// TwinCAT 3 PLC project struckig_unittest
// ProgramVersion: 3.1.4024.12
// libraries:
//   Struckig, * (Struckig)
//   Tc2_Standard, * (Beckhoff Automation GmbH)
//   Tc2_System, * (Beckhoff Automation GmbH)
//   Tc3_Module, * (Beckhoff Automation GmbH)
//   TcUnit, * (www.tcunit.org)
// project tree:
//   / PlcTask.TcTTO (not stored)
//   POUs/ run_and_return_duration.TcPOU, KnownExamplesTest.TcPOU, MAIN.TcPOU
// real-time tasks:
//   TASK PlcTask: cycle T#10ms, priority 20, ADS port 350

// ---- POUs/run_and_return_duration.TcPOU
FUNCTION run_and_return_duration : LREAL
VAR_INPUT
  ruckig : REFERENCE TO Struckig.Ruckig;
  input : REFERENCE TO Struckig.InputParameter;
  output : REFERENCE TO Struckig.OutputParameter;  
END_VAR

WHILE(ruckig.update(input, output) = Struckig.StateEnum.busy)
DO
  input.current_position := output.new_position;
  input.current_velocity := output.new_velocity;
  input.current_acceleration := output.new_acceleration;
END_WHILE

run_and_return_duration := output.trajectory.duration;

END_FUNCTION

// ---- POUs/KnownExamplesTest.TcPOU
FUNCTION_BLOCK KnownExamplesTest EXTENDS TcUnit.FB_TestSuite

example01();
example02();
example03();
example05();
example06();
example07();
example08();
example09();
example10();
example11();
example12();
example13();
example14();
example15();
example16();
example17();
example18();

METHOD example01
VAR_INST
  ruckig : Struckig.Ruckig(0.005);
  input : Struckig.InputParameter(3) := (
    synchronizationType := SynchronizationTypeEnum.none,        
    max_velocity :=         [ 1.0, 1.0, 1.0 ],
    max_acceleration :=     [ 1.0, 1.0, 1.0 ],
    max_jerk :=             [ 1.0, 1.0, 1.0 ],
    current_position :=     [ 0.0, 0.0, 0.0 ],
    current_velocity :=     [ 0.0, 0.0, 0.0 ],
    current_acceleration := [ 0.0, 0.0, 0.0 ],
    target_position :=      [ 0.0, 0.0, 0.0 ],
    target_velocity :=      [ 0.0, 0.0, 0.0 ],
    target_acceleration :=  [ 0.0, 0.0, 0.0 ]
  );
  output : Struckig.OutputParameter;
END_VAR
TEST('Example-01');

AssertEquals_LREAL(Expected := 0.0,
             Actual := run_and_return_duration(ruckig, input, output),
             DELTA := 1E-8,
             Message := '');
 
TEST_FINISHED();
END_METHOD

METHOD example02
VAR_INST
  ruckig : Struckig.Ruckig(0.005);
  input : Struckig.InputParameter(3) := (
    synchronizationType := SynchronizationTypeEnum.none,        
    max_velocity :=         [ 1.0, 1.0, 1.0 ],
    max_acceleration :=     [ 1.0, 1.0, 1.0 ],
    max_jerk :=             [ 1.0, 1.0, 1.0 ],
    current_position :=     [ 0.0, 0.0, 0.0 ],
    current_velocity :=     [ 0.0, 0.0, 0.0 ],
    current_acceleration := [ 0.0, 0.0, 0.0 ],
    target_position :=      [ 0.0, 1E-17, -1E-17 ],
    target_velocity :=      [ 0.0, 0.0, 0.0 ],
    target_acceleration :=  [ 0.0, 0.0, 0.0 ]
  );
  output : Struckig.OutputParameter;  
END_VAR
TEST('Example-02');

AssertEquals_LREAL(Expected := 1E-18,
             Actual := run_and_return_duration(ruckig, input, output),
             Delta := 1E-19,
             Message := '');
 
TEST_FINISHED();
END_METHOD

METHOD example03
VAR_INST
  ruckig : Struckig.Ruckig(0.005);
  input : Struckig.InputParameter(3) := (
    synchronizationType := SynchronizationTypeEnum.none,        
    max_velocity :=         [ 1.0, 1.0, 1.0 ],
    max_acceleration :=     [ 1.0, 1.0, 1.0 ],
    max_jerk :=             [ 1.0, 1.0, 1.0 ],
    current_position :=     [ 0.0, 1E-17, -1E-17 ],
    current_velocity :=     [ 0.0, 0.0, 0.0 ],
    current_acceleration := [ 0.0, 0.0, 0.0 ],
    target_position :=      [ 1.0, 1.0, 1.0 ],
    target_velocity :=      [ 0.0, 0.0, 0.0 ],
    target_acceleration :=  [ 0.0, 0.0, 0.0 ]
  );
  output : Struckig.OutputParameter;
  
END_VAR
TEST('Example-03');

AssertEquals_LREAL(Expected := 3.1748021039,
             Actual := run_and_return_duration(ruckig, input, output),
             DELTA := 1E-8,
             Message := '');
 
TEST_FINISHED();
END_METHOD

METHOD example04
VAR_INST
  ruckig : Struckig.Ruckig(0.005);
  input : Struckig.InputParameter(3) := (
    synchronizationType := SynchronizationTypeEnum.none,        
    max_velocity :=         [ 1.0, 1.0, 1.0 ],
    max_acceleration :=     [ 1.0, 1.0, 1.0 ],
    max_jerk :=             [ 2.0, 2.0, 2.0 ],
    current_position :=     [ 0.0, 0.0, 0.0 ],
    current_velocity :=     [ 0.0, 0.0, 0.0 ],
    current_acceleration := [ 0.0, 0.0, 0.0 ],
    target_position :=      [ 1.0, 1.0, 1.0 ],
    target_velocity :=      [ 0.0, 0.0, 0.0 ],
    target_acceleration :=  [ 0.0, 0.0, 0.0 ]
  );
  output : Struckig.OutputParameter;
  
END_VAR
TEST('Example-04');

AssertEquals_LREAL(Expected := 2.5615528128,
             Actual := run_and_return_duration(ruckig, input, output),
             DELTA := 1E-8,
             Message := '');
 
TEST_FINISHED();
END_METHOD

METHOD example05
VAR_INST
  ruckig : Struckig.Ruckig(0.005);
  input : Struckig.InputParameter(3) := (
    synchronizationType := SynchronizationTypeEnum.none,        
    max_velocity :=         [ 0.6, 0.6, 0.6 ],
    max_acceleration :=     [ 1.0, 1.0, 1.0 ],
    max_jerk :=             [ 2.0, 2.0, 2.0 ],
    current_position :=     [ 0.0, 0.0, 0.0 ],
    current_velocity :=     [ 0.0, 0.0, 0.0 ],
    current_acceleration := [ 0.0, 0.0, 0.0 ],
    target_position :=      [ 1.0, 1.0, 1.0 ],
    target_velocity :=      [ 0.0, 0.0, 0.0 ],
    target_acceleration :=  [ 0.0, 0.0, 0.0 ]
  );
  output : Struckig.OutputParameter;
  
END_VAR
TEST('Example-05');

AssertEquals_LREAL(Expected := 2.7666666667,
             Actual := run_and_return_duration(ruckig, input, output),
             DELTA := 1E-8,
             Message := '');
 
TEST_FINISHED();
END_METHOD

METHOD example06
VAR_INST
  ruckig : Struckig.Ruckig(0.005);
  input : Struckig.InputParameter(3) := (
    synchronizationType := SynchronizationTypeEnum.none,        
    max_velocity :=         [ 0.4, 0.4, 0.4 ],
    max_acceleration :=     [ 1.0, 1.0, 1.0 ],
    max_jerk :=             [ 2.0, 2.0, 2.0 ],
    current_position :=     [ 0.0, 0.0, 0.0 ],
    current_velocity :=     [ 0.0, 0.0, 0.0 ],
    current_acceleration := [ 0.0, 0.0, 0.0 ],
    target_position :=      [ 1.0, 1.0, 1.0 ],
    target_velocity :=      [ 0.0, 0.0, 0.0 ],
    target_acceleration :=  [ 0.0, 0.0, 0.0 ]
  );
  output : Struckig.OutputParameter;
  
END_VAR
TEST('Example-06');

AssertEquals_LREAL(Expected := 3.394427191,
             Actual := run_and_return_duration(ruckig, input, output),
             DELTA := 1E-8,
             Message := '');
 
TEST_FINISHED();
END_METHOD

METHOD example07
VAR_INST
  ruckig : Struckig.Ruckig(0.005);
  input : Struckig.InputParameter(3) := (
    synchronizationType := SynchronizationTypeEnum.none,        
    max_velocity :=         [ 1.0, 1.0, 1.0 ],
    max_acceleration :=     [ 1.0, 1.0, 1.0 ],
    max_jerk :=             [ 2.0, 2.0, 2.0 ],
    current_position :=     [ 0.0, 0.0, 0.0 ],
    current_velocity :=     [ 0.3, 0.3, 0.3 ],
    current_acceleration := [ 0.0, 0.0, 0.0 ],
    target_position :=      [ 1.0, 1.0, 1.0 ],
    target_velocity :=      [ 0.0, 0.0, 0.0 ],
    target_acceleration :=  [ 0.0, 0.0, 0.0 ]
  );
  output : Struckig.OutputParameter;
  
END_VAR
TEST('Example-07');

AssertEquals_LREAL(Expected := 2.2319602829,
             Actual := run_and_return_duration(ruckig, input, output),
             DELTA := 1E-8,
             Message := '');
 
TEST_FINISHED();
END_METHOD

METHOD example08
VAR_INST
  ruckig : Struckig.Ruckig(0.005);
  input : Struckig.InputParameter(3) := (
    synchronizationType := SynchronizationTypeEnum.none,        
    max_velocity :=         [ 0.6, 0.6, 0.6 ],
    max_acceleration :=     [ 1.0, 1.0, 1.0 ],
    max_jerk :=             [ 2.0, 2.0, 2.0 ],
    current_position :=     [ 0.0, 0.0, 0.0 ],
    current_velocity :=     [ 0.3, 0.3, 0.3 ],
    current_acceleration := [ 0.0, 0.0, 0.0 ],
    target_position :=      [ 1.0, 1.0, 1.0 ],
    target_velocity :=      [ 0.0, 0.0, 0.0 ],
    target_acceleration :=  [ 0.0, 0.0, 0.0 ]
  );
  output : Struckig.OutputParameter;
  
END_VAR
TEST('Example-08');

AssertEquals_LREAL(Expected := 2.410315834,
             Actual := run_and_return_duration(ruckig, input, output),
             DELTA := 1E-8,
             Message := '');
 
TEST_FINISHED();
END_METHOD

METHOD example09
VAR_INST
  ruckig : Struckig.Ruckig(0.005);
  input : Struckig.InputParameter(3) := (
    synchronizationType := SynchronizationTypeEnum.none,        
    max_velocity :=         [ 0.6, 0.6, 0.6 ],
    max_acceleration :=     [ 1.0, 1.0, 1.0 ],
    max_jerk :=             [ 2.0, 2.0, 2.0 ],
    current_position :=     [ 0.0, 0.0, 0.0 ],
    current_velocity :=     [ 0.0, 0.0, 0.0 ],
    current_acceleration := [ 0.0, 0.0, 0.0 ],
    target_position :=      [ -1.0, -1.0, -1.0 ],
    target_velocity :=      [ 0.0, 0.0, 0.0 ],
    target_acceleration :=  [ 0.0, 0.0, 0.0 ]
  );
  output : Struckig.OutputParameter;
  
END_VAR
TEST('Example-09');

AssertEquals_LREAL(Expected := 2.7666666667,
             Actual := run_and_return_duration(ruckig, input, output),
             DELTA := 1E-8,
             Message := '');
 
TEST_FINISHED();
END_METHOD

METHOD example10
VAR_INST
  ruckig : Struckig.Ruckig(0.005);
  input : Struckig.InputParameter(3) := (
    synchronizationType := SynchronizationTypeEnum.none,        
    max_velocity :=         [ 10.0, 10.0, 10.0 ],
    max_acceleration :=     [ 10.0, 10.0, 10.0 ],
    max_jerk :=             [ 2.0, 2.0, 2.0 ],
    current_position :=     [ 0.0, 0.0, 0.0 ],
    current_velocity :=     [ 0.2, 0.2, 0.2 ],
    current_acceleration := [ 0.0, 0.0, 0.0 ],
    target_position :=      [ -1.0, -1.0, -1.0 ],
    target_velocity :=      [ 0.0, 0.0, 0.0 ],
    target_acceleration :=  [ 0.0, 0.0, 0.0 ]
  );
  output : Struckig.OutputParameter;
  
END_VAR
TEST('Example-10');

AssertEquals_LREAL(Expected := 2.7338531701,
             Actual := run_and_return_duration(ruckig, input, output),
             DELTA := 1E-8,
             Message := '');
 
TEST_FINISHED();
END_METHOD

METHOD example11
VAR_INST
  ruckig : Struckig.Ruckig(0.005);
  input : Struckig.InputParameter(3) := (
    synchronizationType := SynchronizationTypeEnum.none,        
    max_velocity :=         [ 0.4, 0.4, 0.4 ],
    max_acceleration :=     [ 1.0, 1.0, 1.0 ],
    max_jerk :=             [ 2.0, 2.0, 2.0 ],
    current_position :=     [ -1.0, -1.0, -1.0 ],
    current_velocity :=     [ 0.2, 0.2, 0.2 ],
    current_acceleration := [ 0.0, 0.0, 0.0 ],
    target_position :=      [ 1.0, 1.0, 1.0 ],
    target_velocity :=      [ 0.0, 0.0, 0.0 ],
    target_acceleration :=  [ 0.0, 0.0, 0.0 ]
  );
  output : Struckig.OutputParameter;
  
END_VAR
TEST('Example-11');

AssertEquals_LREAL(Expected := 5.6053274785,
             Actual := run_and_return_duration(ruckig, input, output),
             DELTA := 1E-8,
             Message := '');
 
TEST_FINISHED();
END_METHOD

METHOD example12
VAR_INST
  ruckig : Struckig.Ruckig(0.005);
  input : Struckig.InputParameter(3) := (
    synchronizationType := SynchronizationTypeEnum.none,        
    max_velocity :=         [ 3.0, 3.0, 3.0 ],
    max_acceleration :=     [ 0.5, 0.5, 0.5 ],
    max_jerk :=             [ 0.2, 0.2, 0.2 ],
    current_position :=     [ 0.3888899206957 - 10E-14, 0.0, 0.0 ],
    current_velocity :=     [ 0.2231429352410215, 0.0, 0.0 ],
    current_acceleration := [ -0.2987593916455, 0.0, 0.0 ],
    target_position :=      [ 0.5, 0.0, 0.0 ],
    target_velocity :=      [ 0.0, 0.0, 0.0 ],
    target_acceleration :=  [ 0.0, 0.0, 0.0 ]
  );
  output : Struckig.OutputParameter;
  
END_VAR
TEST('Example-12');

AssertEquals_LREAL(Expected := 1.4939456041,
             Actual := run_and_return_duration(ruckig, input, output),
             DELTA := 1E-8,
             Message := '');
 
TEST_FINISHED();
END_METHOD

METHOD example13
VAR_INST
  ruckig : Struckig.Ruckig(0.005);
  input : Struckig.InputParameter(3) := (
    synchronizationType := SynchronizationTypeEnum.none,        
    max_velocity :=         [ 12.9892953062198, 3.74169932927481, 1.42398447457303 ],
    max_acceleration :=     [ 4.2162106624246, 10.2906731766853, 2.1869079548297 ],
    max_jerk :=             [ 8.03496976453435, 0.200684346397485 - 1.0E-14, 0.0848503482861296 ],
    current_position :=     [ -5.54640573838539, -2.34195463203842, 5.10070661762967 ],
    current_velocity :=     [ 0.824843228617216, -1.03863337183304, -0.749451523227729 ],
    current_acceleration := [ -0.119403564898501, 0.923861820607788, 3.04022341347259 ],
    target_position :=      [ -1.58293112753888, 0.383405919465141, 5.79349604610299 ],
    target_velocity :=      [ -1.59453676324393, 0.0, -0.0693173526513803 ],
    target_acceleration :=  [ -0.664429703711622, 0.0, 0.0 ]
  );
  output : Struckig.OutputParameter;
  
END_VAR
TEST('Example-13');

AssertEquals_LREAL(Expected := 1921.0797627836,
             Actual := run_and_return_duration(ruckig, input, output),
             DELTA := 1E-8,
             Message := '');
 
TEST_FINISHED();
END_METHOD

METHOD example14
VAR_INST
  ruckig : Struckig.Ruckig(0.005);
  input : Struckig.InputParameter(3) := (
    synchronizationType := SynchronizationTypeEnum.none,        
    max_velocity :=         [ 8.65978706670502, 5.94921088330542, 10.7652253566829 ],
    max_acceleration :=     [ 3.40137210377608, 4.04166318018487, 10.8617860610581 ],
    max_jerk :=             [ 10.9542353113865, 3.11056302676629, 0.798055744482636 + 9e-12 ],
    current_position :=     [ -6.49539540831446, 6.14883133273172, -2.02636240900911 ],
    current_velocity :=     [ -1.14327601654428, 0.00991019970085593, -1.00932863927626 ],
    current_acceleration := [ -1.73501068960131, -0.584885092422228, 0 ],
    target_position :=      [ 4.4676187540058, 2.93367894961155, -0.646008452514058 ],
    target_velocity :=      [ -0.544559915133859, 0.298517792372943, 1.6058847848484 ],
    target_acceleration :=  [ -1.31832055647831, 0, 0 ]
  );
  output : Struckig.OutputParameter;
  
END_VAR
TEST('Example-14');

AssertEquals_LREAL(Expected := 4.6277455678,
             Actual := run_and_return_duration(ruckig, input, output),
             DELTA := 1E-8,
             Message := '');
 
TEST_FINISHED();
END_METHOD

METHOD example15
VAR_INST
  ruckig : Struckig.Ruckig(0.005);
  input : Struckig.InputParameter(3) := (
    synchronizationType := SynchronizationTypeEnum.none,        
    max_velocity :=         [ 7.97399137456765, 2.68591430972239, 9.54987666746364 ],
    max_acceleration :=     [ 5.44679859206862, 7.61752909348119, 0.473482772614085 ],
    max_jerk :=             [ 7.88958080921515, 5.26855927512131, 0.764061581326592 - 1e-14 ],
    current_position :=     [ 7.06378251402596, -2.4834697862831, -0.843847405371359 ],
    current_velocity :=     [ 0.436985859305842, 0.0708113515655622, -0.751266816040307 ],
    current_acceleration := [ -0.80835350359544, 0, -0.355284934641626 ],
    target_position :=      [ 4.40606827118048, -2.84629921001043, -2.91829890043522 ],
    target_velocity :=      [ 0.555084596169823, 0, -1.24631524923535 ],
    target_acceleration :=  [ 0.463000173872542, 0, 0 ]
  );
  output : Struckig.OutputParameter;
  
END_VAR
TEST('Example-15');

AssertEquals_LREAL(Expected := 8.8739464323,
             Actual := run_and_return_duration(ruckig, input, output),
             DELTA := 1E-8,
             Message := '');
 
TEST_FINISHED();
END_METHOD

METHOD example16
VAR_INST
  ruckig : Struckig.Ruckig(0.005);
  input : Struckig.InputParameter(3) := (
    synchronizationType := SynchronizationTypeEnum.none,        
    max_velocity :=         [ 0.1241065584614779, 1, 1 ],
    max_acceleration :=     [ 1.808598147153279, 1, 1 ],
    max_jerk :=             [ 2.516849090900998 - 3e-15, 1, 1 ],
    current_position :=     [ -7.962737259350095, 0, 0 ],
    current_velocity :=     [ -0.8844863500141733, 0, 0 ],
    current_acceleration := [ 2.252932547031004, 0, 0 ],
    target_position :=      [ -3.547368989678775, 0, 0 ],
    target_velocity :=      [ 0, 0, 0 ],
    target_acceleration :=  [ 0.217242176687843, 0, 0 ]
  );
  output : Struckig.OutputParameter;
  
END_VAR
TEST('Example-16');

AssertEquals_LREAL(Expected := 38.3409477609,
             Actual := run_and_return_duration(ruckig, input, output),
             DELTA := 1E-8,
             Message := '');
 
TEST_FINISHED();
END_METHOD

METHOD example17
VAR_INST
  ruckig : Struckig.Ruckig(0.005);
  input : Struckig.InputParameter(3) := (
    synchronizationType := SynchronizationTypeEnum.none,    
    max_velocity :=         [ 1.863775561344568, 0.4357836109021987, 6.260907804906162 ],
    max_acceleration :=     [ 9.49223908896113, 9.002562577262177, 1.119142029086944 ],
    max_jerk :=             [ 8.689575453772798, 0.09322235504216797, 0.1594452521517275 + 3e-15 ],
    current_position :=     [ -4.180150148354134, 1.030371049895473, -2.660154279239869 ],
    current_velocity :=     [ 1.673805463302308, -1.435796222257198, 0.9711306630275642 ],
    current_acceleration := [ 1.412175048500792, 1.892262449040863, -1.128847905860926 ],
    target_position :=      [ 2.079913937916431, 1.839862681333277, 2.341421542126605 ],
    target_velocity :=      [ 0.7537566830764975, 0, 0.02507782261105568 ],
    target_acceleration :=  [ -0.8610296259045267, -0.07876324073516261, 0 ]
  );
  output : Struckig.OutputParameter;
  
END_VAR
TEST('Example-17');

AssertEquals_LREAL(Expected := 1135.0135089249,
             Actual := run_and_return_duration(ruckig, input, output),
             DELTA := 1E-8,
             Message := '');
 
TEST_FINISHED();
END_METHOD

METHOD example18
VAR_INST
  ruckig : Struckig.Ruckig(0.005);
  input : Struckig.InputParameter(3) := (
    synchronizationType := SynchronizationTypeEnum.none,
    max_velocity :=         [ 6.144314006624488, 2.93258338415229, 0.1820021269527196 ],
    max_acceleration :=     [ 5.199401036221791, 1.848176490768948, 11.11168017805234 ],
    max_jerk :=             [ 9.940940357283978, 10.46997753899755, 0.08166297169205029 ],
    current_position :=     [ -4.490717417930574, 3.467236624628543, -0.7545929089757601 ],
    current_velocity :=     [ 0.1839756723363622, -0.4356283320280516, 0.7490399525818022 ],
    current_acceleration := [ -1.057769973808928, 0, -2.368645439140517 ],
    target_position :=      [ -4.928244836531066, -4.821780824003112, -8.20567952461017 ],
    target_velocity :=      [ 0.1097319156272965, -0.9272874846270881, 0 ],
    target_acceleration :=  [ 0.03089046366221739, -0.9744054582899561, 0 ]
  );
  output : Struckig.OutputParameter;
  
END_VAR
TEST('Example-18');

AssertEquals_LREAL(Expected := 7295.4375633935,
             Actual := run_and_return_duration(ruckig, input, output),
             DELTA := 1E-8,
             Message := '');
 
TEST_FINISHED();
END_METHOD

END_FUNCTION_BLOCK

// ---- POUs/MAIN.TcPOU
PROGRAM MAIN
VAR
  knownExamplesTest : KnownExamplesTest;  
END_VAR

TcUnit.RUN();

END_PROGRAM
